(* PLC project Unnamed, Unknown Unnamed 1 *)
(* stored: creationDateTime 2023-03-23T15:04:11, modificationDateTime 2023-03-24T22:41:34 *)

PROGRAM SEVEN_SEGMENT_DISPLAY
  VAR_INPUT
    W : BOOL := 0;
    X : BOOL := 0;
    Y : BOOL := 0;
    Z : BOOL := 0;
  END_VAR
  VAR_IN_OUT
    A : BOOL;
  END_VAR
  VAR_OUTPUT
    B : BOOL;
    C : BOOL;
    DD : BOOL;
    EE : BOOL;
    F : BOOL;
    G : BOOL;
  END_VAR
  VAR  (* added by the conversion: wires and edge detectors of the diagram *)
    _NOT18_OUT : BOOL;
    _NOT17_OUT : BOOL;
    _NOT16_OUT : BOOL;
    _OR24_OUT : BOOL;
  END_VAR

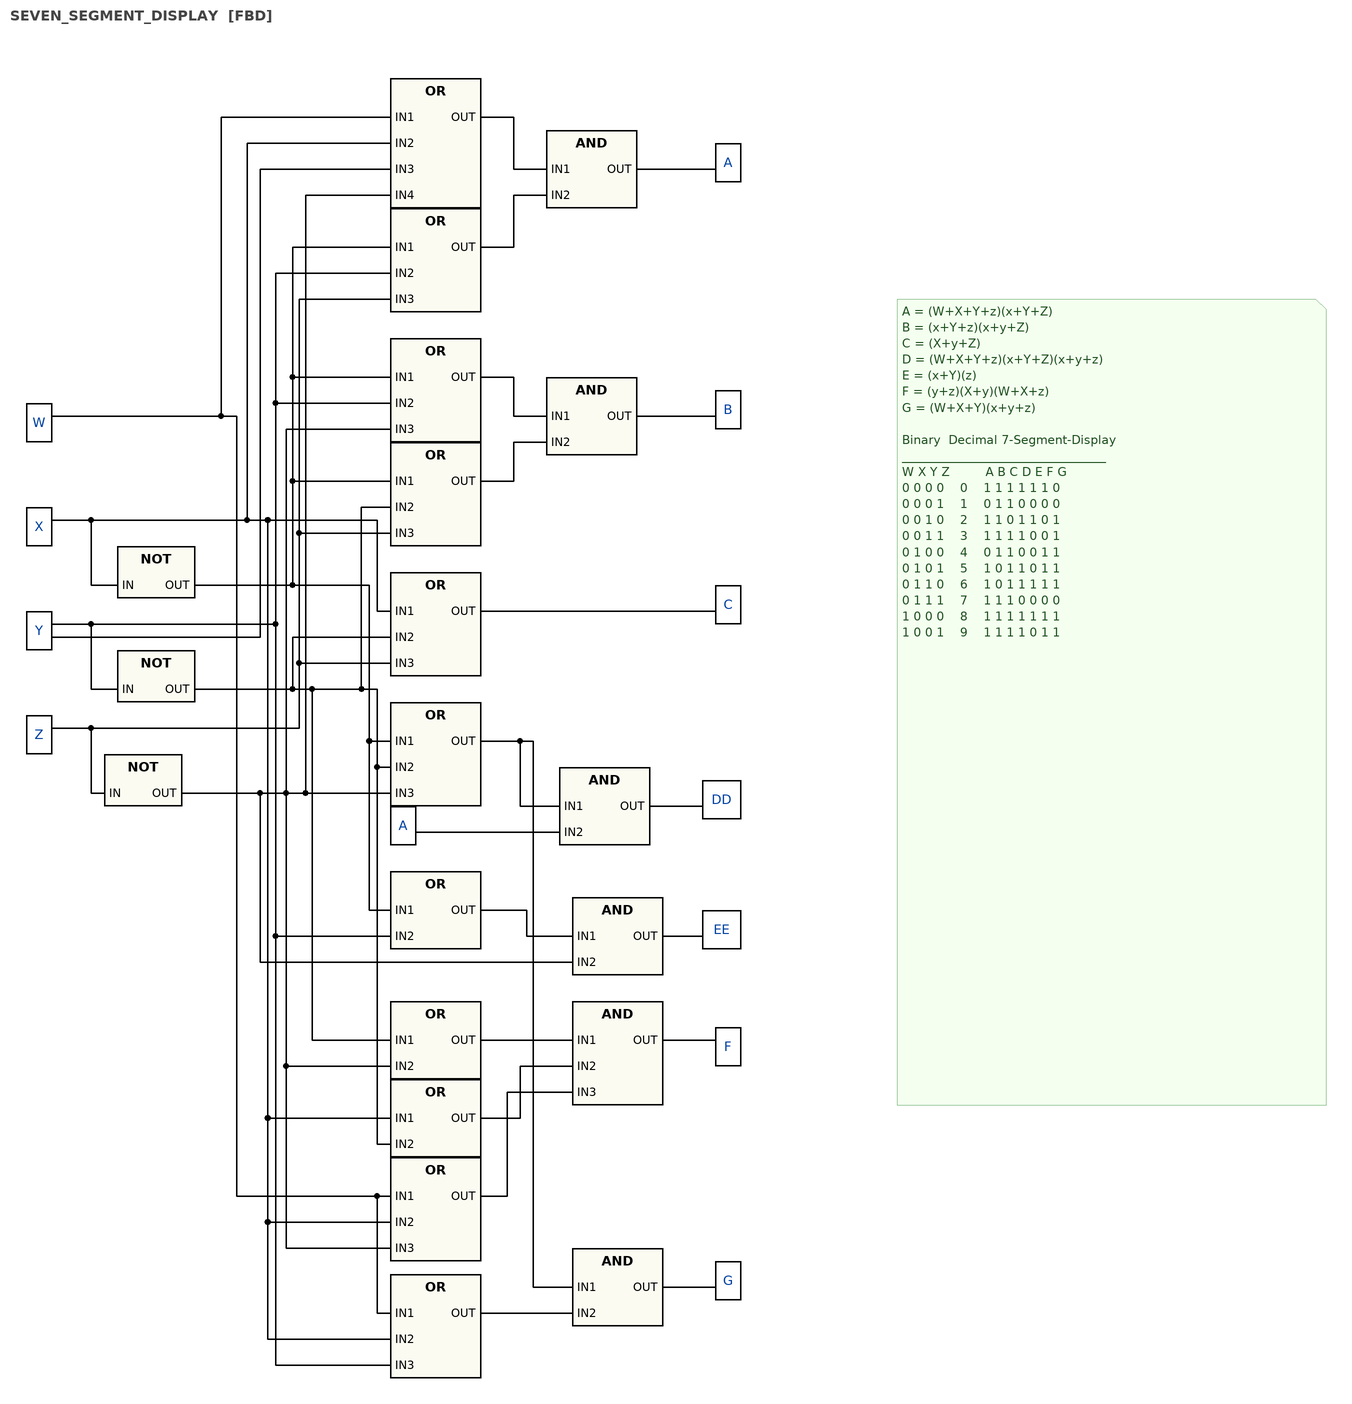
(* FBD diagram, written out as Structured Text *)
_NOT18_OUT := NOT Z;
_NOT17_OUT := NOT X;
A := (W OR X OR Y OR _NOT18_OUT) AND (_NOT17_OUT OR Y OR Z);
(* A = (W+X+Y+z)(x+Y+Z)
B = (x+Y+z)(x+y+Z)
C = (X+y+Z)
D = (W+X+Y+z)(x+Y+Z)(x+y+z)
E = (x+Y)(z)
F = (y+z)(X+y)(W+X+z)
G = (W+X+Y)(x+y+z)

Binary  Decimal 7-Segment-Display
__________________________________
W X Y Z         A B C D E F G  
0 0 0 0    0    1 1 1 1 1 1 0
0 0 0 1    1    0 1 1 0 0 0 0
0 0 1 0    2    1 1 0 1 1 0 1
0 0 1 1    3    1 1 1 1 0 0 1
0 1 0 0    4    0 1 1 0 0 1 1
0 1 0 1    5    1 0 1 1 0 1 1
0 1 1 0    6    1 0 1 1 1 1 1
0 1 1 1    7    1 1 1 0 0 0 0
1 0 0 0    8    1 1 1 1 1 1 1
1 0 0 1    9    1 1 1 1 0 1 1 *)
_NOT16_OUT := NOT Y;
B := (_NOT17_OUT OR Y OR _NOT18_OUT) AND (_NOT17_OUT OR _NOT16_OUT OR Z);
C := X OR _NOT16_OUT OR Z;
_OR24_OUT := _NOT17_OUT OR _NOT16_OUT OR _NOT18_OUT;
DD := _OR24_OUT AND A;
EE := (_NOT17_OUT OR Y) AND _NOT18_OUT;
F := (_NOT16_OUT OR _NOT18_OUT) AND (X OR _NOT16_OUT) AND (W OR X OR _NOT18_OUT);
G := _OR24_OUT AND (W OR X OR Y);
END_PROGRAM

CONFIGURATION Config0
  RESOURCE Res0 ON PLC
    TASK task0(INTERVAL := T#20ms, PRIORITY := 0);
    PROGRAM instance0 WITH task0 : SEVEN_SEGMENT_DISPLAY;
  END_RESOURCE
END_CONFIGURATION
